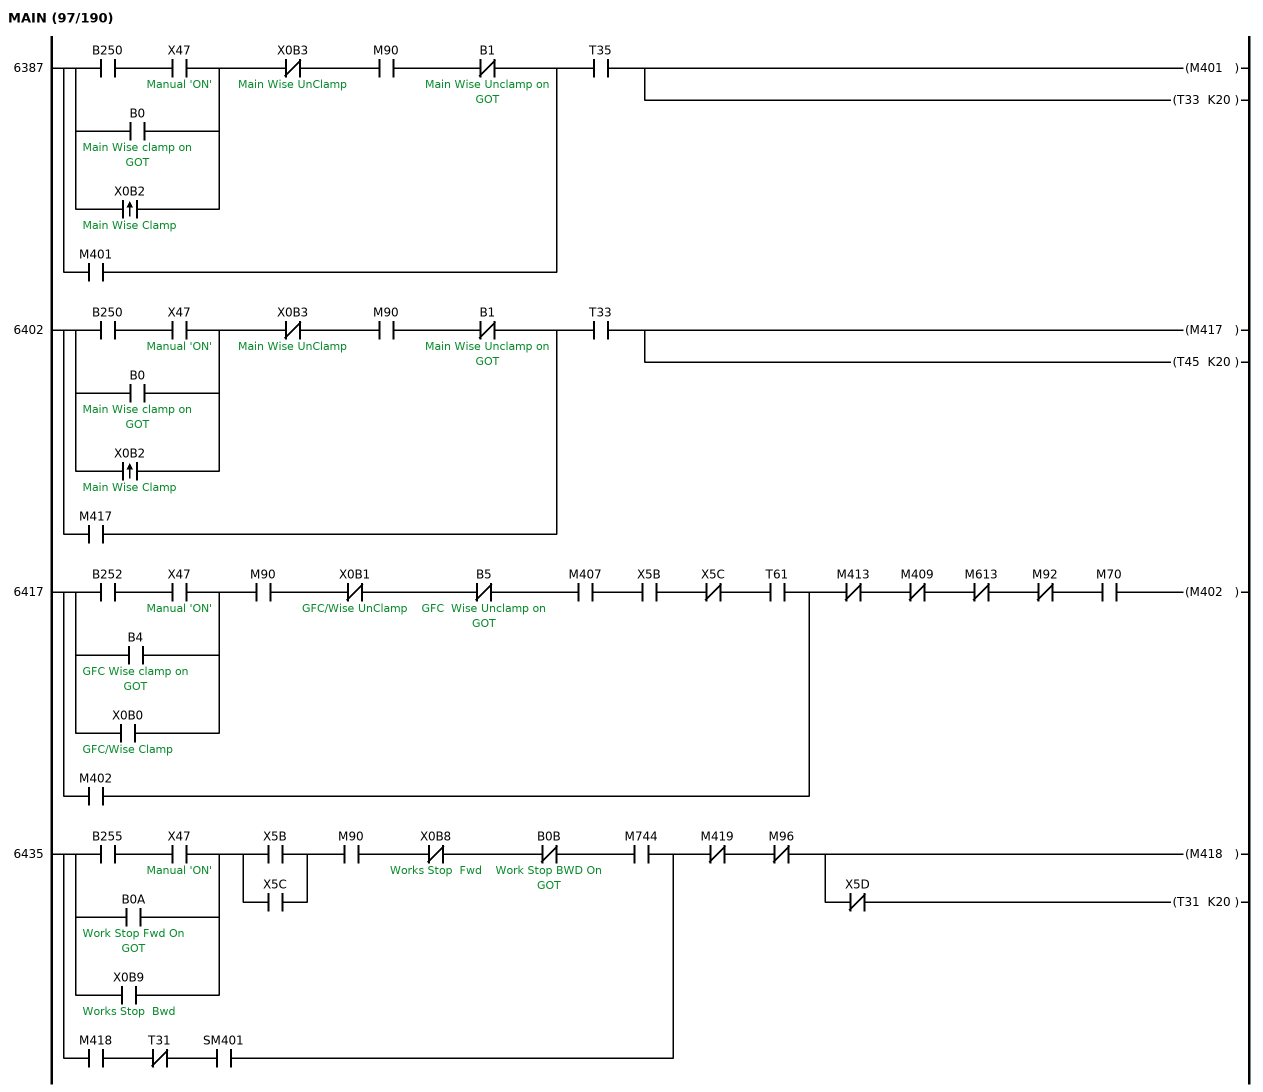
[picture p96: ladder of MAIN, rungs at steps 6387 to 6435]
6387  LD      B250
      AND     X47  ; Manual 'ON'
      OR      B0  ; Main Wise clamp on GOT
      ORP     X0B2  ; Main Wise Clamp
      ANI     X0B3  ; Main Wise UnClamp
      AND     M90
      ANI     B1  ; Main Wise Unclamp on GOT
      OR      M401
      AND     T35
      OUT     M401
      OUT     T33 K20
6402  LD      B250
      AND     X47  ; Manual 'ON'
      OR      B0  ; Main Wise clamp on GOT
      ORP     X0B2  ; Main Wise Clamp
      ANI     X0B3  ; Main Wise UnClamp
      AND     M90
      ANI     B1  ; Main Wise Unclamp on GOT
      OR      M417
      AND     T33
      OUT     M417
      OUT     T45 K20
6417  LD      B252
      AND     X47  ; Manual 'ON'
      OR      B4  ; GFC Wise clamp on GOT
      OR      X0B0  ; GFC/Wise Clamp
      AND     M90
      ANI     X0B1  ; GFC/Wise UnClamp
      ANI     B5  ; GFC  Wise Unclamp on GOT
      AND     M407
      AND     X5B
      ANI     X5C
      AND     T61
      OR      M402
      ANI     M413
      ANI     M409
      ANI     M613
      ANI     M92
      AND     M70
      OUT     M402
6435  LD      B255
      AND     X47  ; Manual 'ON'
      OR      B0A  ; Work Stop Fwd On GOT
      OR      X0B9  ; Works Stop  Bwd
      LD      X5B
      OR      X5C
      ANB
      AND     M90
      ANI     X0B8  ; Works Stop  Fwd
      ANI     B0B  ; Work Stop BWD On GOT
      AND     M744
      LD      M418
      ANI     T31
      AND     SM401
      ORB
      ANI     M419
      ANI     M96
      OUT     M418
      ANI     X5D
      OUT     T31 K20
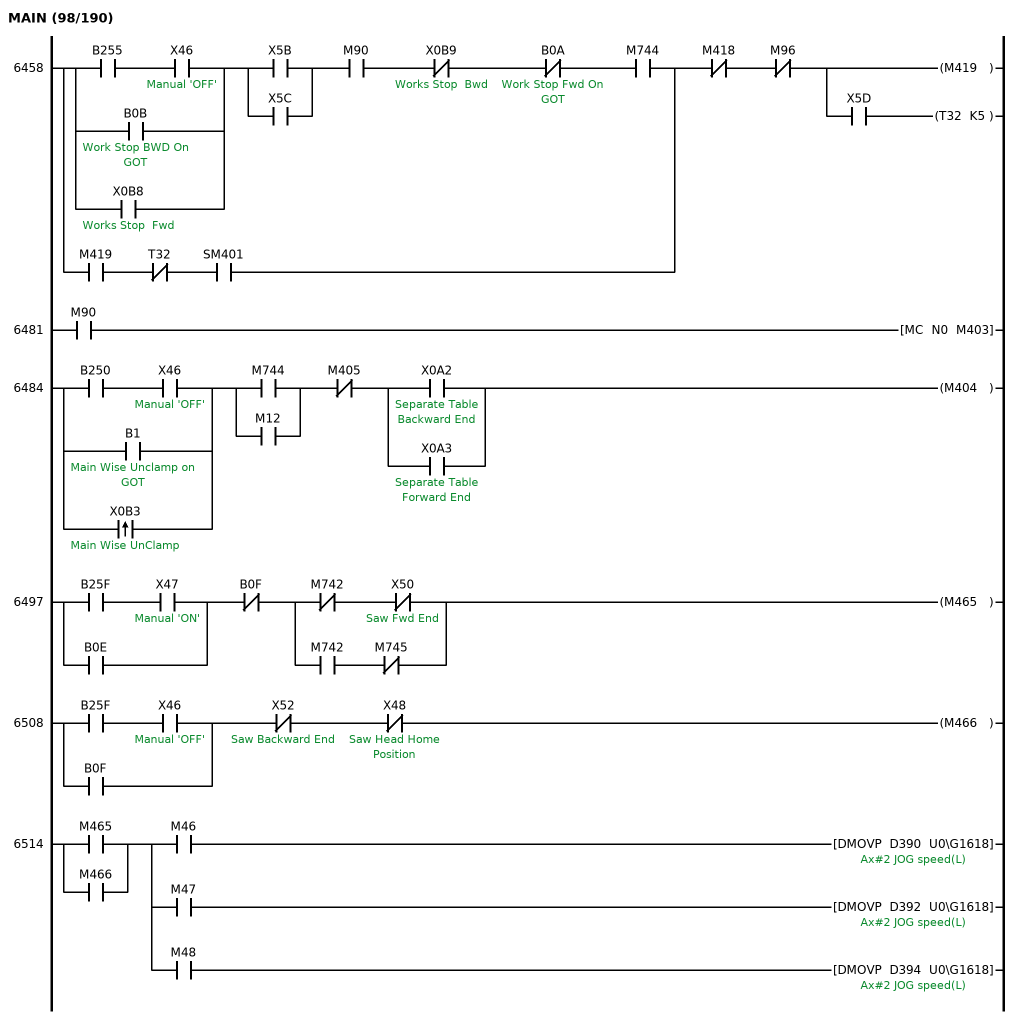
6458  LD      B255
      AND     X46  ; Manual 'OFF'
      OR      B0B  ; Work Stop BWD On GOT
      OR      X0B8  ; Works Stop  Fwd
      LD      X5B
      OR      X5C
      ANB
      AND     M90
      ANI     X0B9  ; Works Stop  Bwd
      ANI     B0A  ; Work Stop Fwd On GOT
      AND     M744
      LD      M419
      ANI     T32
      AND     SM401
      ORB
      ANI     M418
      ANI     M96
      OUT     M419
      AND     X5D
      OUT     T32 K5
6481  LD      M90
      MC      N0 M403
6484  LD      B250
      AND     X46  ; Manual 'OFF'
      OR      B1  ; Main Wise Unclamp on GOT
      ORP     X0B3  ; Main Wise UnClamp
      LD      M744
      OR      M12
      ANB
      ANI     M405
      LD      X0A2  ; Separate Table Backward End
      OR      X0A3  ; Separate Table Forward End
      ANB
      OUT     M404
6497  LD      B25F
      AND     X47  ; Manual 'ON'
      OR      B0E
      ANI     B0F
      LDI     M742
      ANI     X50  ; Saw Fwd End
      LD      M742
      ANI     M745
      ORB
      ANB
      OUT     M465
6508  LD      B25F
      AND     X46  ; Manual 'OFF'
      OR      B0F
      ANI     X52  ; Saw Backward End
      ANI     X48  ; Saw Head Home Position
      OUT     M466
6514  LD      M465
      OR      M466
      MPS
      AND     M46
      DMOVP   D390 U0\G1618
      MRD
      AND     M47
      DMOVP   D392 U0\G1618
      MPP
      AND     M48
      DMOVP   D394 U0\G1618
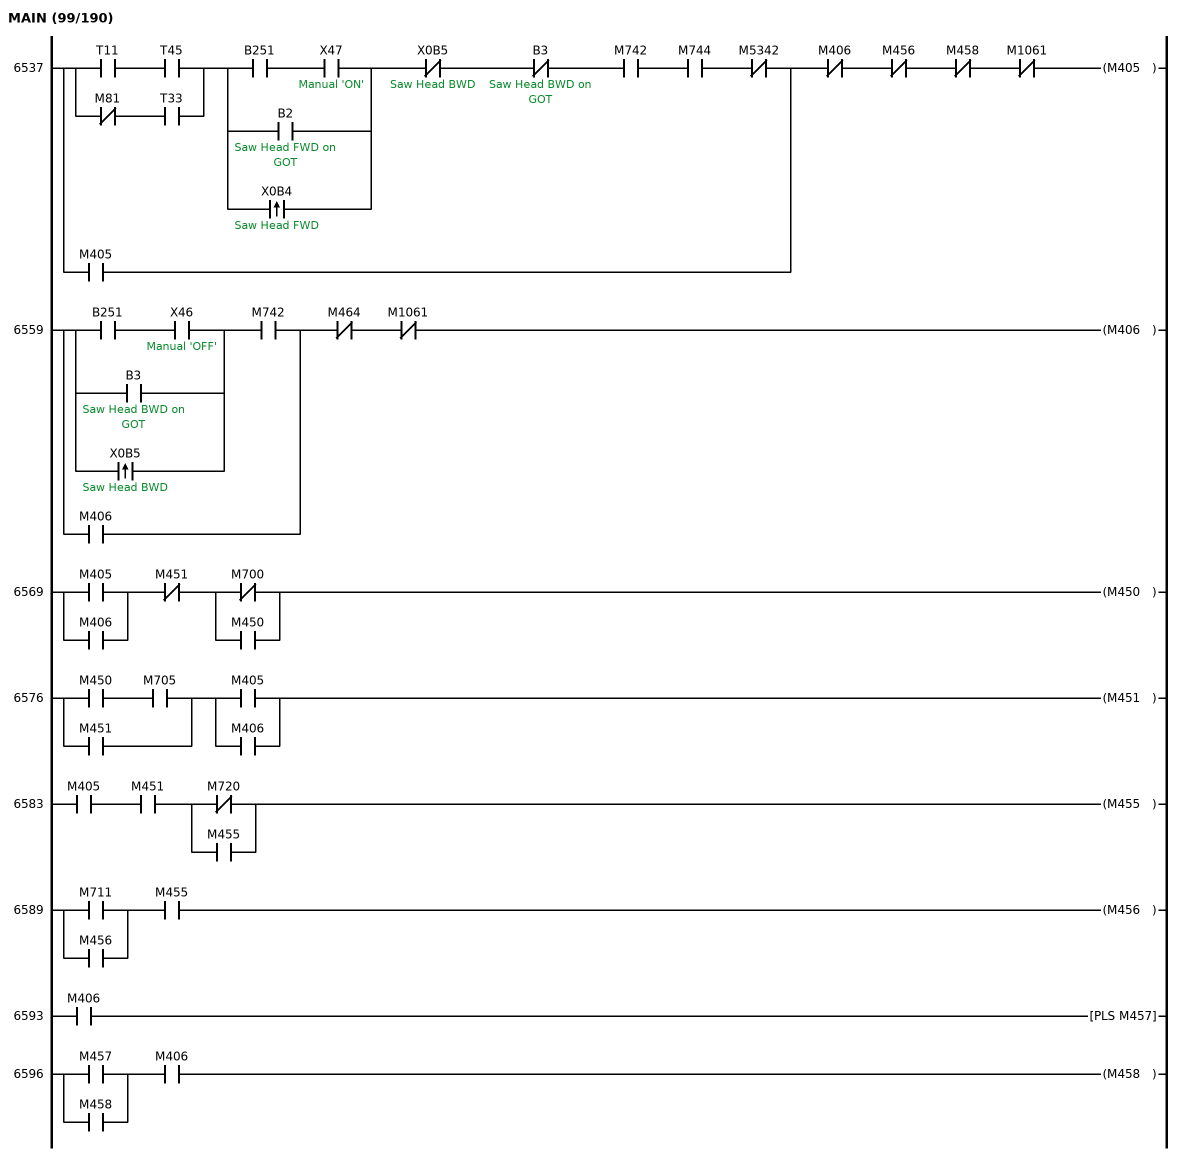
6537  LD      T11
      AND     T45
      LDI     M81
      AND     T33
      ORB
      LD      B251
      AND     X47  ; Manual 'ON'
      OR      B2  ; Saw Head FWD on GOT
      ORP     X0B4  ; Saw Head FWD
      ANB
      ANI     X0B5  ; Saw Head BWD
      ANI     B3  ; Saw Head BWD on GOT
      AND     M742
      AND     M744
      ANI     M5342
      OR      M405
      ANI     M406
      ANI     M456
      ANI     M458
      ANI     M1061
      OUT     M405
6559  LD      B251
      AND     X46  ; Manual 'OFF'
      OR      B3  ; Saw Head BWD on GOT
      ORP     X0B5  ; Saw Head BWD
      AND     M742
      OR      M406
      ANI     M464
      ANI     M1061
      OUT     M406
6569  LD      M405
      OR      M406
      ANI     M451
      LDI     M700
      OR      M450
      ANB
      OUT     M450
6576  LD      M450
      AND     M705
      OR      M451
      LD      M405
      OR      M406
      ANB
      OUT     M451
6583  LD      M405
      AND     M451
      LDI     M720
      OR      M455
      ANB
      OUT     M455
6589  LD      M711
      OR      M456
      AND     M455
      OUT     M456
6593  LD      M406
      PLS     M457
6596  LD      M457
      OR      M458
      AND     M406
      OUT     M458
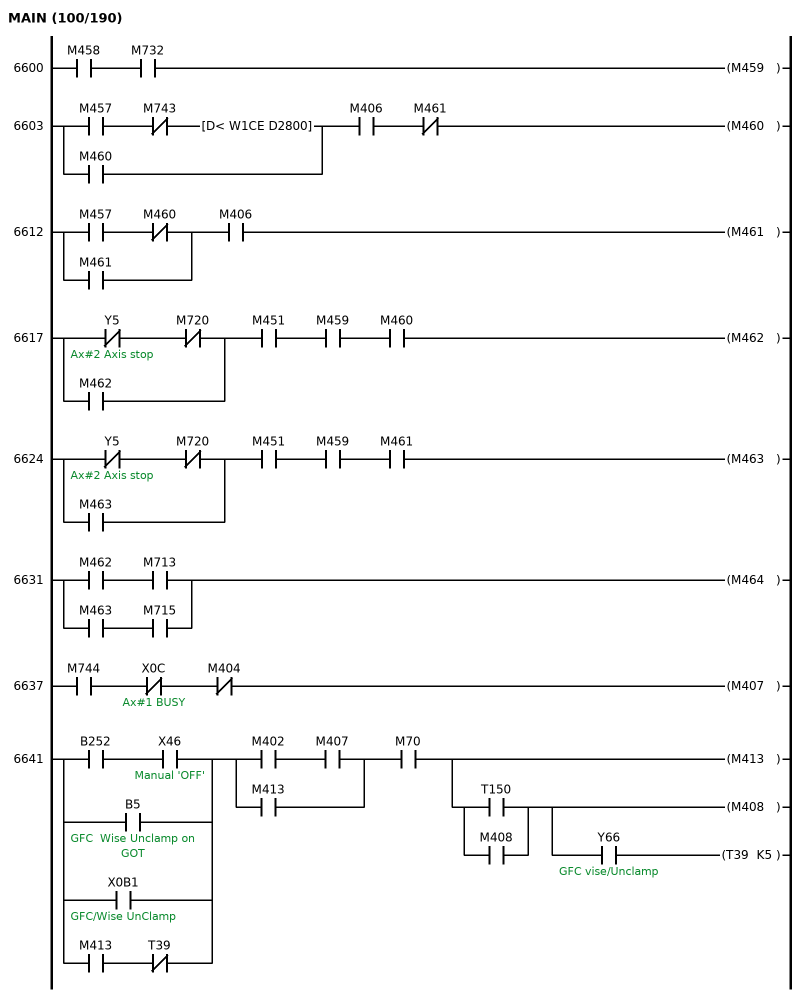
6600  LD      M458
      AND     M732
      OUT     M459
6603  LD      M457
      ANI     M743
      ANDD<   W1CE D2800
      OR      M460
      AND     M406
      ANI     M461
      OUT     M460
6612  LD      M457
      ANI     M460
      OR      M461
      AND     M406
      OUT     M461
6617  LDI     Y5  ; Ax#2 Axis stop
      ANI     M720
      OR      M462
      AND     M451
      AND     M459
      AND     M460
      OUT     M462
6624  LDI     Y5  ; Ax#2 Axis stop
      ANI     M720
      OR      M463
      AND     M451
      AND     M459
      AND     M461
      OUT     M463
6631  LD      M462
      AND     M713
      LD      M463
      AND     M715
      ORB
      OUT     M464
6637  LD      M744
      ANI     X0C  ; Ax#1 BUSY
      ANI     M404
      OUT     M407
6641  LD      B252
      AND     X46  ; Manual 'OFF'
      OR      B5  ; GFC  Wise Unclamp on GOT
      OR      X0B1  ; GFC/Wise UnClamp
      LD      M413
      ANI     T39
      ORB
      LD      M402
      AND     M407
      OR      M413
      ANB
      AND     M70
      OUT     M413
      LD      T150
      OR      M408
      ANB
      OUT     M408
      AND     Y66  ; GFC vise/Unclamp
      OUT     T39 K5
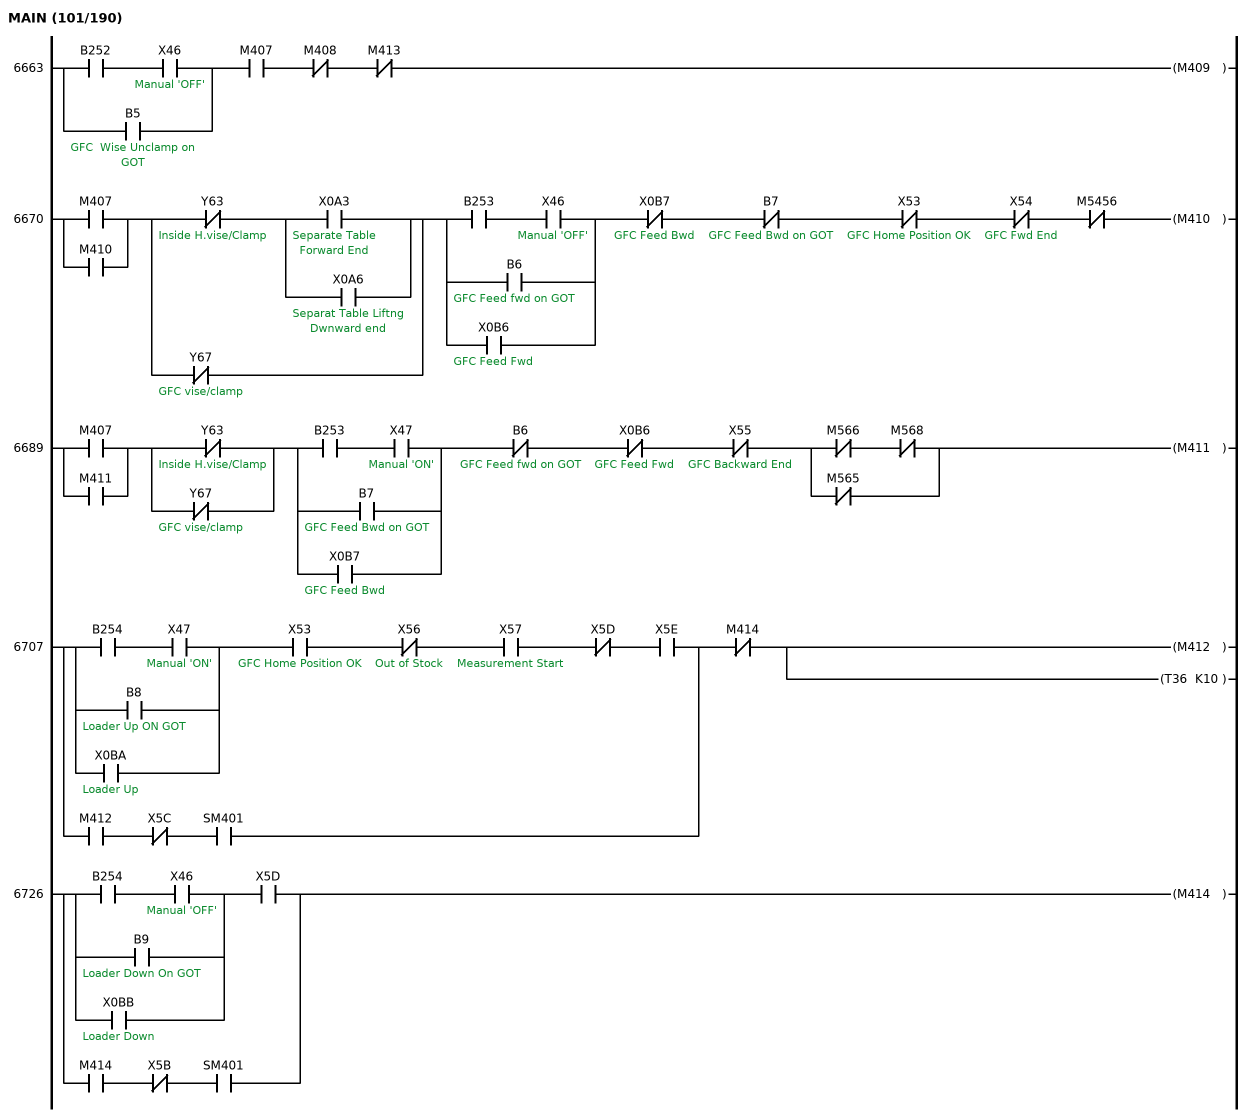
6663  LD      B252
      AND     X46  ; Manual 'OFF'
      OR      B5  ; GFC  Wise Unclamp on GOT
      AND     M407
      ANI     M408
      ANI     M413
      OUT     M409
6670  LD      M407
      OR      M410
      LDI     Y63  ; Inside H.vise/Clamp
      LD      X0A3  ; Separate Table Forward End
      OR      X0A6  ; Separat Table Liftng Dwnward end
      ANB
      ORI     Y67  ; GFC vise/clamp
      ANB
      LD      B253
      AND     X46  ; Manual 'OFF'
      OR      B6  ; GFC Feed fwd on GOT
      OR      X0B6  ; GFC Feed Fwd
      ANB
      ANI     X0B7  ; GFC Feed Bwd
      ANI     B7  ; GFC Feed Bwd on GOT
      ANI     X53  ; GFC Home Position OK
      ANI     X54  ; GFC Fwd End
      ANI     M5456
      OUT     M410
6689  LD      M407
      OR      M411
      LDI     Y63  ; Inside H.vise/Clamp
      ORI     Y67  ; GFC vise/clamp
      ANB
      LD      B253
      AND     X47  ; Manual 'ON'
      OR      B7  ; GFC Feed Bwd on GOT
      OR      X0B7  ; GFC Feed Bwd
      ANB
      ANI     B6  ; GFC Feed fwd on GOT
      ANI     X0B6  ; GFC Feed Fwd
      ANI     X55  ; GFC Backward End
      LDI     M566
      ANI     M568
      ORI     M565
      ANB
      OUT     M411
6707  LD      B254
      AND     X47  ; Manual 'ON'
      OR      B8  ; Loader Up ON GOT
      OR      X0BA  ; Loader Up
      AND     X53  ; GFC Home Position OK
      ANI     X56  ; Out of Stock
      AND     X57  ; Measurement Start
      ANI     X5D
      AND     X5E
      LD      M412
      ANI     X5C
      AND     SM401
      ORB
      ANI     M414
      OUT     M412
      OUT     T36 K10
6726  LD      B254
      AND     X46  ; Manual 'OFF'
      OR      B9  ; Loader Down On GOT
      OR      X0BB  ; Loader Down
      AND     X5D
      LD      M414
      ANI     X5B
      AND     SM401
      ORB
      OUT     M414
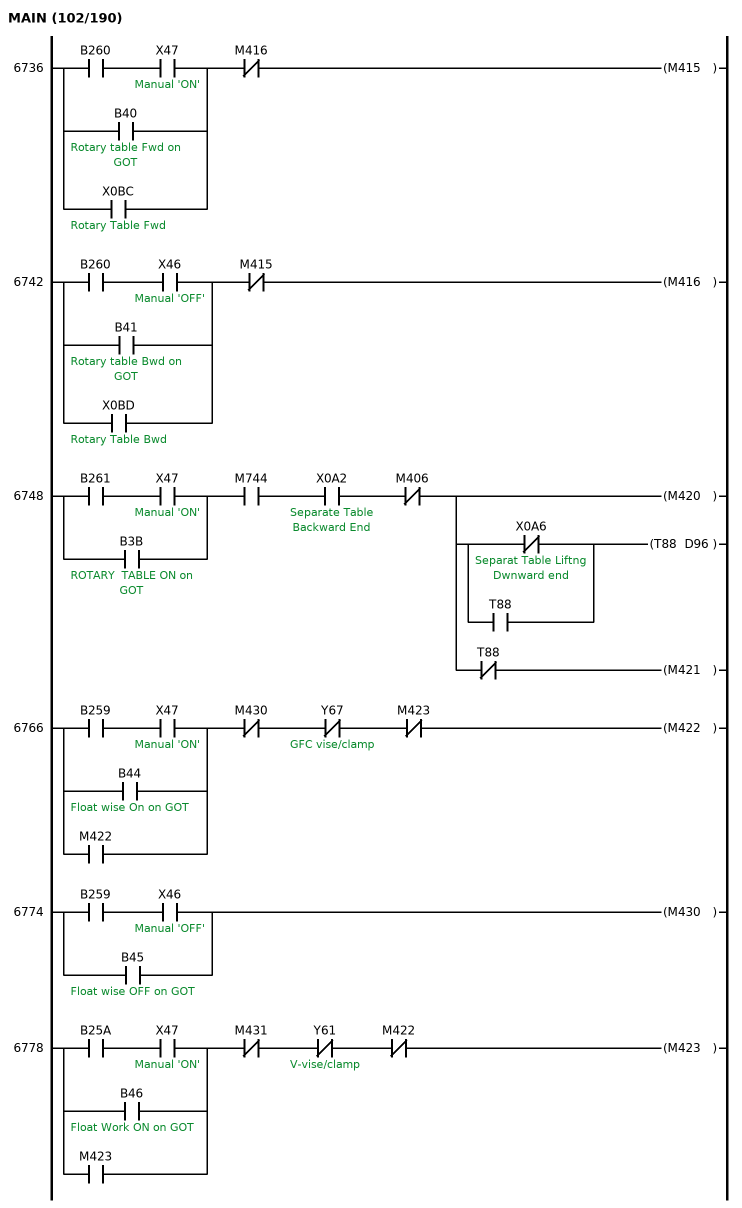
6736  LD      B260
      AND     X47  ; Manual 'ON'
      OR      B40  ; Rotary table Fwd on GOT
      OR      X0BC  ; Rotary Table Fwd
      ANI     M416
      OUT     M415
6742  LD      B260
      AND     X46  ; Manual 'OFF'
      OR      B41  ; Rotary table Bwd on GOT
      OR      X0BD  ; Rotary Table Bwd
      ANI     M415
      OUT     M416
6748  LD      B261
      AND     X47  ; Manual 'ON'
      OR      B3B  ; ROTARY  TABLE ON on GOT
      AND     M744
      AND     X0A2  ; Separate Table Backward End
      ANI     M406
      OUT     M420
      MPS
      LDI     X0A6  ; Separat Table Liftng Dwnward end
      OR      T88
      ANB
      OUT     T88 D96
      MPP
      ANI     T88
      OUT     M421
6766  LD      B259
      AND     X47  ; Manual 'ON'
      OR      B44  ; Float wise On on GOT
      OR      M422
      ANI     M430
      ANI     Y67  ; GFC vise/clamp
      ANI     M423
      OUT     M422
6774  LD      B259
      AND     X46  ; Manual 'OFF'
      OR      B45  ; Float wise OFF on GOT
      OUT     M430
6778  LD      B25A
      AND     X47  ; Manual 'ON'
      OR      B46  ; Float Work ON on GOT
      OR      M423
      ANI     M431
      ANI     Y61  ; V-vise/clamp
      ANI     M422
      OUT     M423
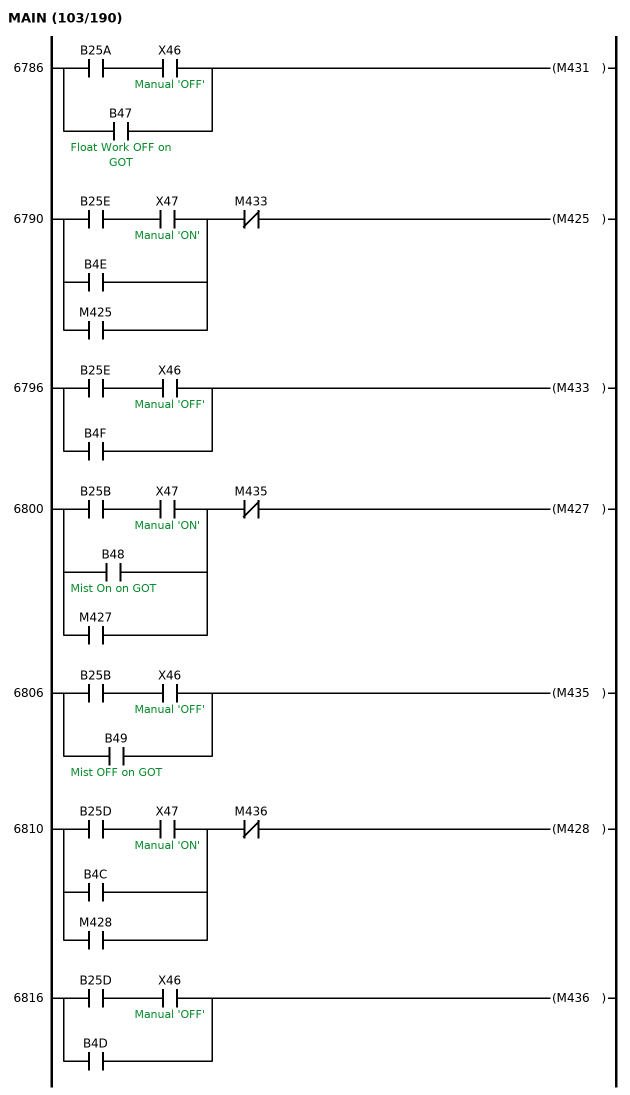
6786  LD      B25A
      AND     X46  ; Manual 'OFF'
      OR      B47  ; Float Work OFF on GOT
      OUT     M431
6790  LD      B25E
      AND     X47  ; Manual 'ON'
      OR      B4E
      OR      M425
      ANI     M433
      OUT     M425
6796  LD      B25E
      AND     X46  ; Manual 'OFF'
      OR      B4F
      OUT     M433
6800  LD      B25B
      AND     X47  ; Manual 'ON'
      OR      B48  ; Mist On on GOT
      OR      M427
      ANI     M435
      OUT     M427
6806  LD      B25B
      AND     X46  ; Manual 'OFF'
      OR      B49  ; Mist OFF on GOT
      OUT     M435
6810  LD      B25D
      AND     X47  ; Manual 'ON'
      OR      B4C
      OR      M428
      ANI     M436
      OUT     M428
6816  LD      B25D
      AND     X46  ; Manual 'OFF'
      OR      B4D
      OUT     M436
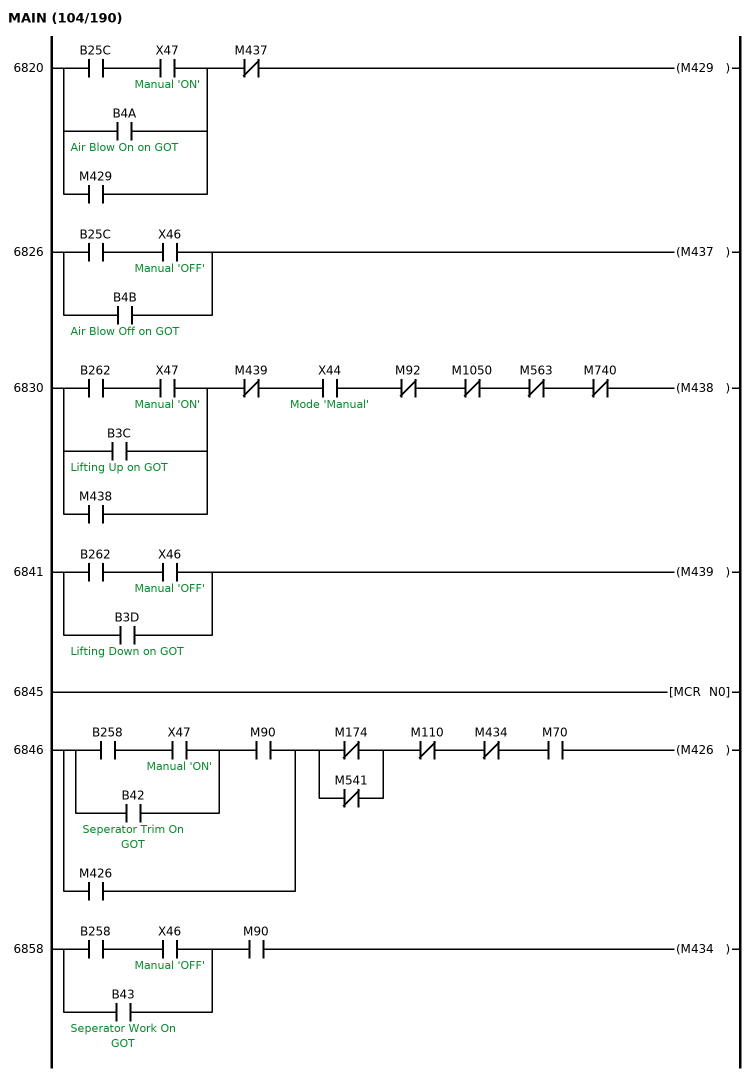
6820  LD      B25C
      AND     X47  ; Manual 'ON'
      OR      B4A  ; Air Blow On on GOT
      OR      M429
      ANI     M437
      OUT     M429
6826  LD      B25C
      AND     X46  ; Manual 'OFF'
      OR      B4B  ; Air Blow Off on GOT
      OUT     M437
6830  LD      B262
      AND     X47  ; Manual 'ON'
      OR      B3C  ; Lifting Up on GOT
      OR      M438
      ANI     M439
      AND     X44  ; Mode 'Manual'
      ANI     M92
      ANI     M1050
      ANI     M563
      ANI     M740
      OUT     M438
6841  LD      B262
      AND     X46  ; Manual 'OFF'
      OR      B3D  ; Lifting Down on GOT
      OUT     M439
6845  MCR     N0
6846  LD      B258
      AND     X47  ; Manual 'ON'
      OR      B42  ; Seperator Trim On GOT
      AND     M90
      OR      M426
      LDI     M174
      ORI     M541
      ANB
      ANI     M110
      ANI     M434
      AND     M70
      OUT     M426
6858  LD      B258
      AND     X46  ; Manual 'OFF'
      OR      B43  ; Seperator Work On GOT
      AND     M90
      OUT     M434
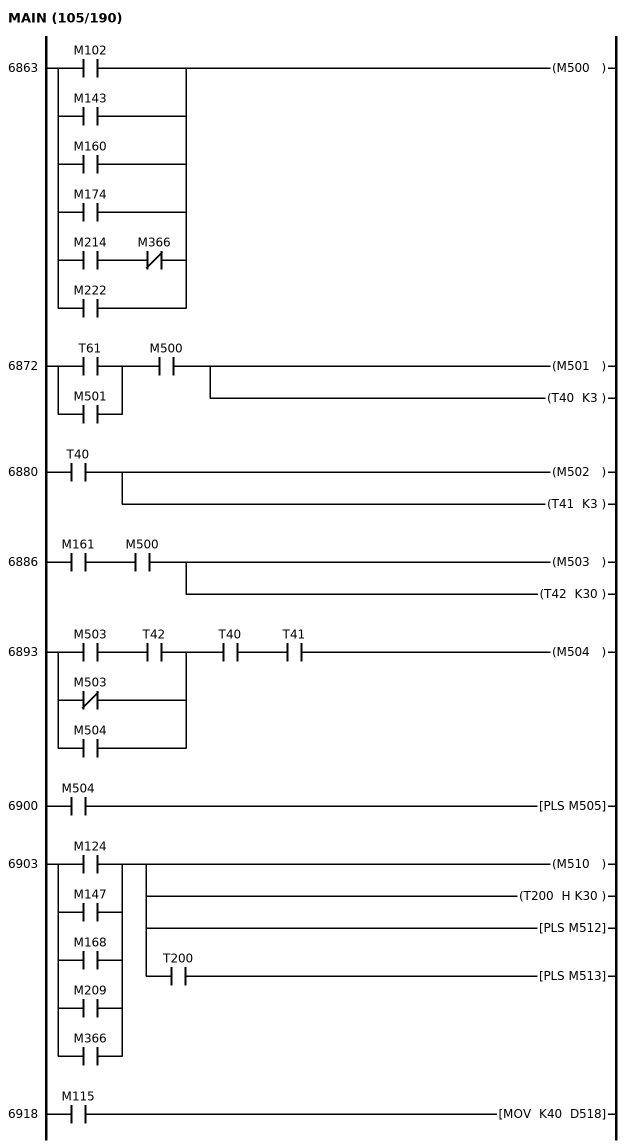
6863  LD      M102
      OR      M143
      OR      M160
      OR      M174
      LD      M214
      ANI     M366
      ORB
      OR      M222
      OUT     M500
6872  LD      T61
      OR      M501
      AND     M500
      OUT     M501
      OUT     T40 K3
6880  LD      T40
      OUT     M502
      OUT     T41 K3
6886  LD      M161
      AND     M500
      OUT     M503
      OUT     T42 K30
6893  LD      M503
      AND     T42
      ORI     M503
      OR      M504
      AND     T40
      AND     T41
      OUT     M504
6900  LD      M504
      PLS     M505
6903  LD      M124
      OR      M147
      OR      M168
      OR      M209
      OR      M366
      OUT     M510
      OUTH    T200 K30
      PLS     M512
      AND     T200
      PLS     M513
6918  LD      M115
      MOV     K40 D518
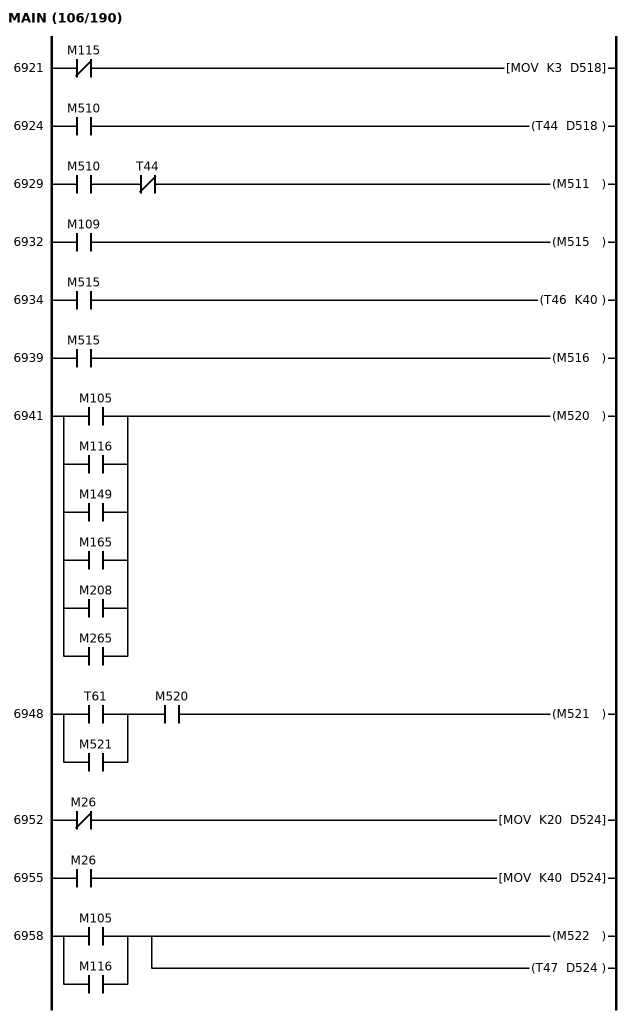
6921  LDI     M115
      MOV     K3 D518
6924  LD      M510
      OUT     T44 D518
6929  LD      M510
      ANI     T44
      OUT     M511
6932  LD      M109
      OUT     M515
6934  LD      M515
      OUT     T46 K40
6939  LD      M515
      OUT     M516
6941  LD      M105
      OR      M116
      OR      M149
      OR      M165
      OR      M208
      OR      M265
      OUT     M520
6948  LD      T61
      OR      M521
      AND     M520
      OUT     M521
6952  LDI     M26
      MOV     K20 D524
6955  LD      M26
      MOV     K40 D524
6958  LD      M105
      OR      M116
      OUT     M522
      OUT     T47 D524
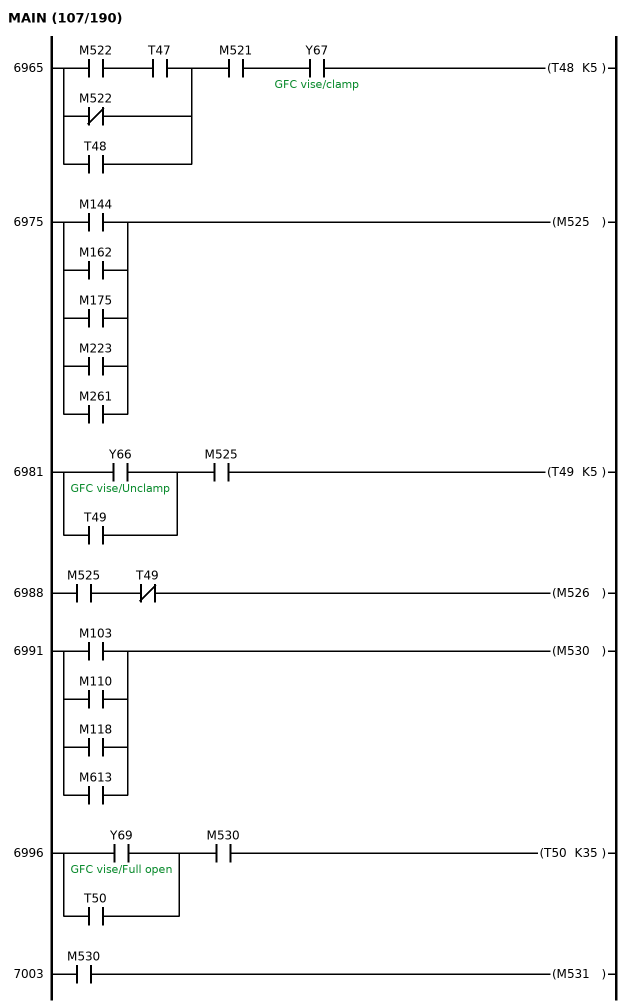
6965  LD      M522
      AND     T47
      ORI     M522
      OR      T48
      AND     M521
      AND     Y67  ; GFC vise/clamp
      OUT     T48 K5
6975  LD      M144
      OR      M162
      OR      M175
      OR      M223
      OR      M261
      OUT     M525
6981  LD      Y66  ; GFC vise/Unclamp
      OR      T49
      AND     M525
      OUT     T49 K5
6988  LD      M525
      ANI     T49
      OUT     M526
6991  LD      M103
      OR      M110
      OR      M118
      OR      M613
      OUT     M530
6996  LD      Y69  ; GFC vise/Full open
      OR      T50
      AND     M530
      OUT     T50 K35
7003  LD      M530
      OUT     M531
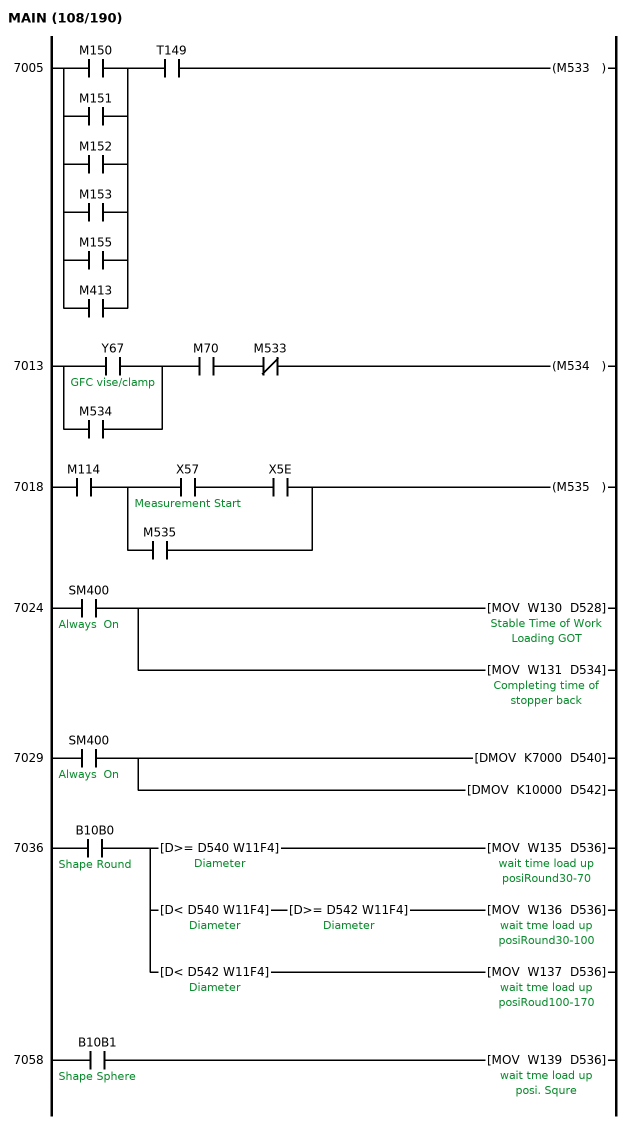
7005  LD      M150
      OR      M151
      OR      M152
      OR      M153
      OR      M155
      OR      M413
      AND     T149
      OUT     M533
7013  LD      Y67  ; GFC vise/clamp
      OR      M534
      AND     M70
      ANI     M533
      OUT     M534
7018  LD      M114
      LD      X57  ; Measurement Start
      AND     X5E
      OR      M535
      ANB
      OUT     M535
7024  LD      SM400  ; Always  On
      MOV     W130 D528
      MOV     W131 D534  ; Completing time of stopper back
7029  LD      SM400  ; Always  On
      DMOV    K7000 D540
      DMOV    K10000 D542
7036  LD      B10B0  ; Shape Round
      MPS
      ANDD>=  D540 W11F4  ; Diameter
      MOV     W135 D536  ; wait time load up posiRound30-70
      MRD
      ANDD<   D540 W11F4  ; Diameter
      ANDD>=  D542 W11F4  ; Diameter
      MOV     W136 D536  ; wait tme load up posiRound30-100
      MPP
      ANDD<   D542 W11F4  ; Diameter
      MOV     W137 D536  ; wait tme load up posiRoud100-170
7058  LD      B10B1  ; Shape Sphere
      MOV     W139 D536  ; wait tme load up posi. Squre
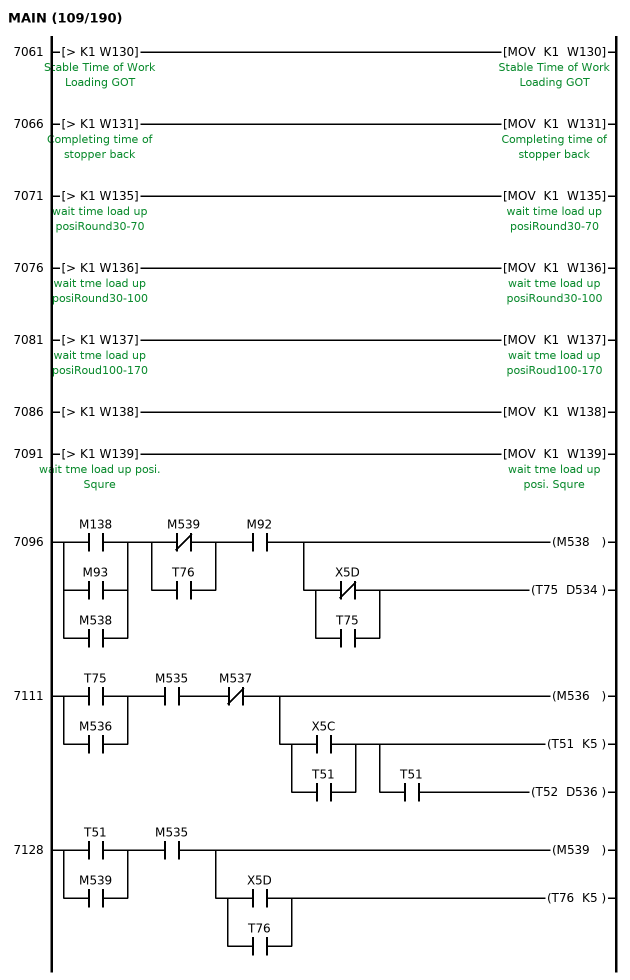
7061  LD>     K1 W130  ; Stable Time of Work Loading GOT
      MOV     K1 W130
7066  LD>     K1 W131  ; Completing time of stopper back
      MOV     K1 W131
7071  LD>     K1 W135  ; wait time load up posiRound30-70
      MOV     K1 W135
7076  LD>     K1 W136  ; wait tme load up posiRound30-100
      MOV     K1 W136
7081  LD>     K1 W137  ; wait tme load up posiRoud100-170
      MOV     K1 W137
7086  LD>     K1 W138
      MOV     K1 W138
7091  LD>     K1 W139  ; wait tme load up posi. Squre
      MOV     K1 W139
7096  LD      M138
      OR      M93
      OR      M538
      LDI     M539
      OR      T76
      ANB
      AND     M92
      OUT     M538
      LDI     X5D
      OR      T75
      ANB
      OUT     T75 D534
7111  LD      T75
      OR      M536
      AND     M535
      ANI     M537
      OUT     M536
      LD      X5C
      OR      T51
      ANB
      OUT     T51 K5
      AND     T51
      OUT     T52 D536
7128  LD      T51
      OR      M539
      AND     M535
      OUT     M539
      LD      X5D
      OR      T76
      ANB
      OUT     T76 K5
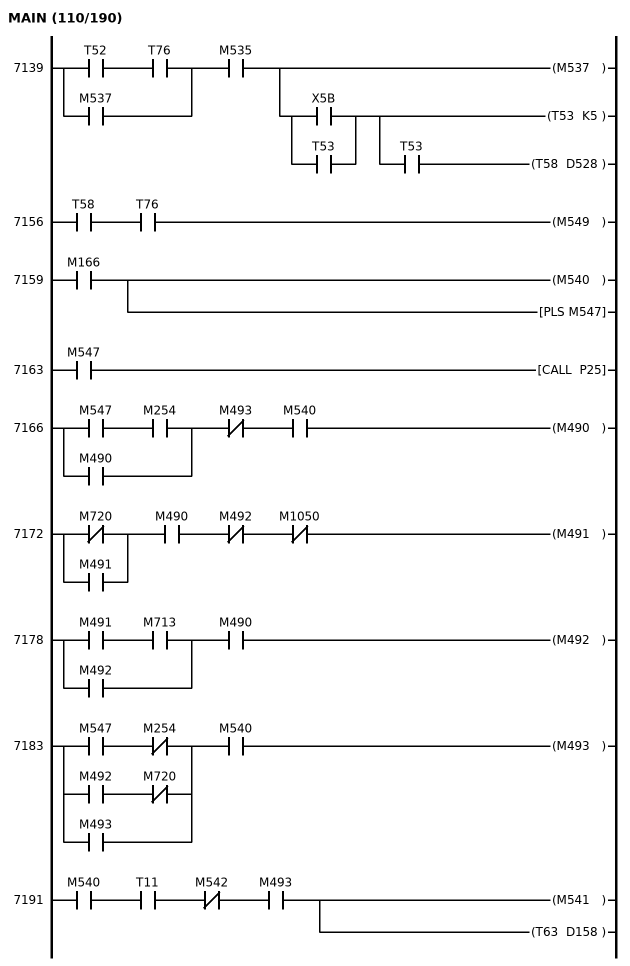
7139  LD      T52
      AND     T76
      OR      M537
      AND     M535
      OUT     M537
      LD      X5B
      OR      T53
      ANB
      OUT     T53 K5
      AND     T53
      OUT     T58 D528
7156  LD      T58
      AND     T76
      OUT     M549
7159  LD      M166
      OUT     M540
      PLS     M547
7163  LD      M547
      CALL    P25
7166  LD      M547
      AND     M254
      OR      M490
      ANI     M493
      AND     M540
      OUT     M490
7172  LDI     M720
      OR      M491
      AND     M490
      ANI     M492
      ANI     M1050
      OUT     M491
7178  LD      M491
      AND     M713
      OR      M492
      AND     M490
      OUT     M492
7183  LD      M547
      ANI     M254
      LD      M492
      ANI     M720
      ORB
      OR      M493
      AND     M540
      OUT     M493
7191  LD      M540
      AND     T11
      ANI     M542
      AND     M493
      OUT     M541
      OUT     T63 D158
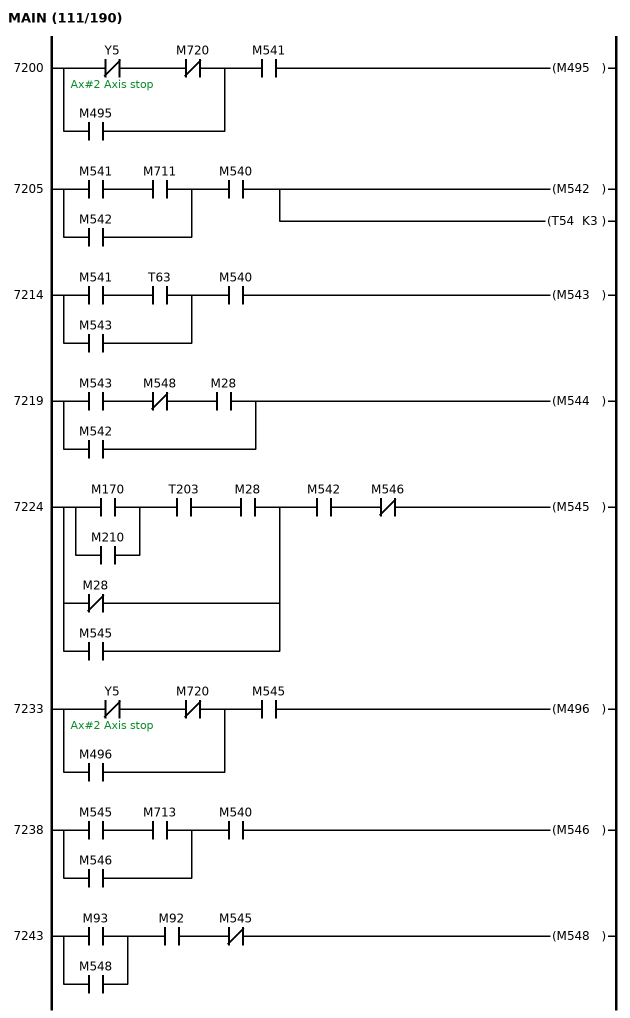
7200  LDI     Y5  ; Ax#2 Axis stop
      ANI     M720
      OR      M495
      AND     M541
      OUT     M495
7205  LD      M541
      AND     M711
      OR      M542
      AND     M540
      OUT     M542
      OUT     T54 K3
7214  LD      M541
      AND     T63
      OR      M543
      AND     M540
      OUT     M543
7219  LD      M543
      ANI     M548
      AND     M28
      OR      M542
      OUT     M544
7224  LD      M170
      OR      M210
      AND     T203
      AND     M28
      ORI     M28
      OR      M545
      AND     M542
      ANI     M546
      OUT     M545
7233  LDI     Y5  ; Ax#2 Axis stop
      ANI     M720
      OR      M496
      AND     M545
      OUT     M496
7238  LD      M545
      AND     M713
      OR      M546
      AND     M540
      OUT     M546
7243  LD      M93
      OR      M548
      AND     M92
      ANI     M545
      OUT     M548
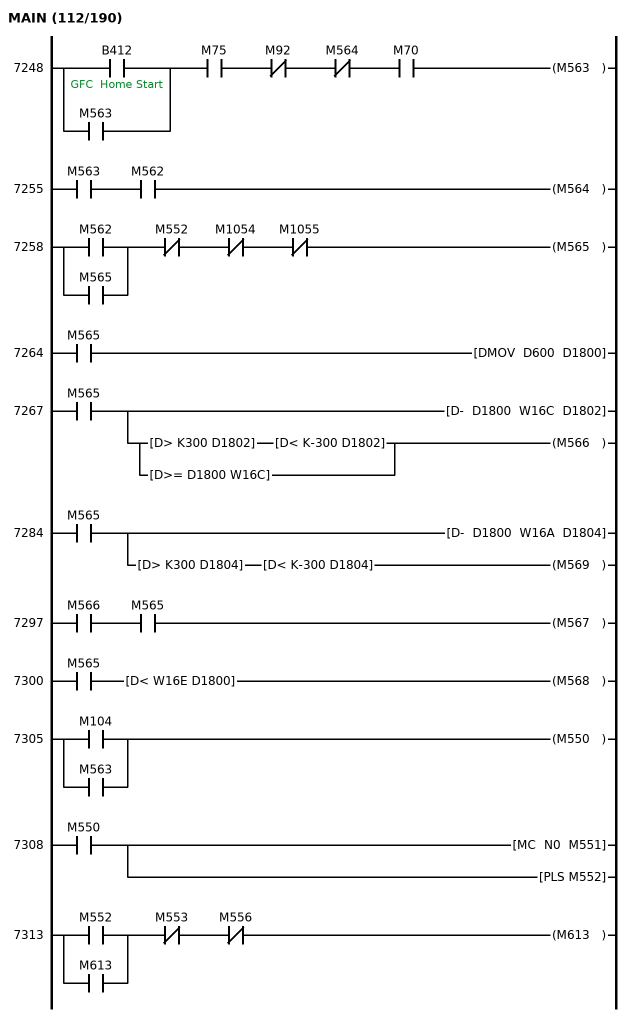
7248  LD      B412  ; GFC  Home Start
      OR      M563
      AND     M75
      ANI     M92
      ANI     M564
      AND     M70
      OUT     M563
7255  LD      M563
      AND     M562
      OUT     M564
7258  LD      M562
      OR      M565
      ANI     M552
      ANI     M1054
      ANI     M1055
      OUT     M565
7264  LD      M565
      DMOV    D600 D1800
7267  LD      M565
      D-      D1800 W16C D1802
      LDD>    K300 D1802
      ANDD<   K-300 D1802
      ORD>=   D1800 W16C
      ANB
      OUT     M566
7284  LD      M565
      D-      D1800 W16A D1804
      ANDD>   K300 D1804
      ANDD<   K-300 D1804
      OUT     M569
7297  LD      M566
      AND     M565
      OUT     M567
7300  LD      M565
      ANDD<   W16E D1800
      OUT     M568
7305  LD      M104
      OR      M563
      OUT     M550
7308  LD      M550
      MC      N0 M551
      PLS     M552
7313  LD      M552
      OR      M613
      ANI     M553
      ANI     M556
      OUT     M613
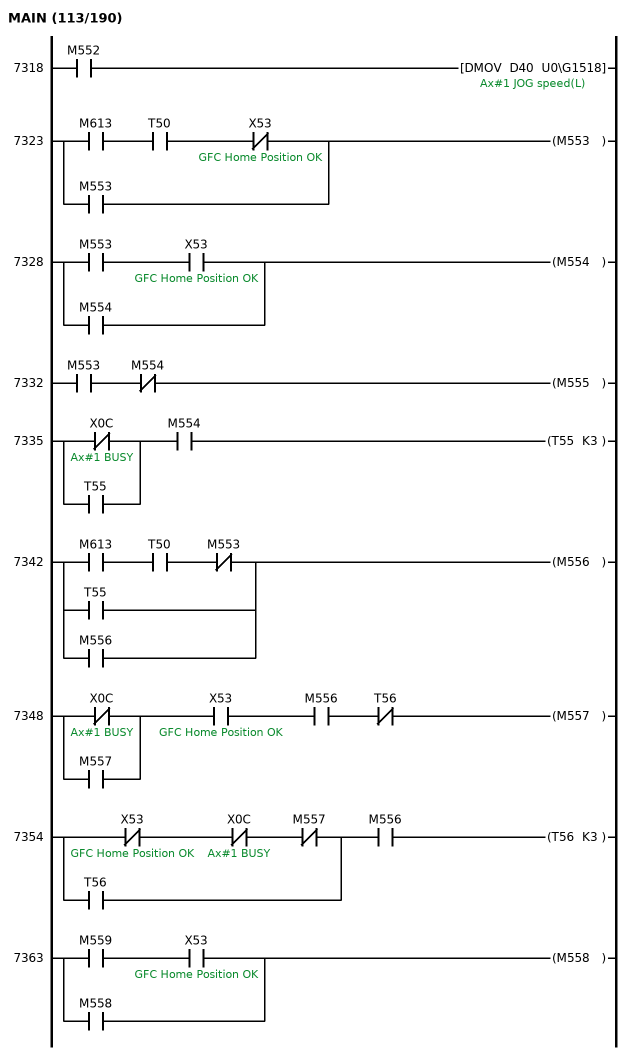
7318  LD      M552
      DMOV    D40 U0\G1518
7323  LD      M613
      AND     T50
      ANI     X53  ; GFC Home Position OK
      OR      M553
      OUT     M553
7328  LD      M553
      AND     X53  ; GFC Home Position OK
      OR      M554
      OUT     M554
7332  LD      M553
      ANI     M554
      OUT     M555
7335  LDI     X0C  ; Ax#1 BUSY
      OR      T55
      AND     M554
      OUT     T55 K3
7342  LD      M613
      AND     T50
      ANI     M553
      OR      T55
      OR      M556
      OUT     M556
7348  LDI     X0C  ; Ax#1 BUSY
      OR      M557
      AND     X53  ; GFC Home Position OK
      AND     M556
      ANI     T56
      OUT     M557
7354  LDI     X53  ; GFC Home Position OK
      ANI     X0C  ; Ax#1 BUSY
      ANI     M557
      OR      T56
      AND     M556
      OUT     T56 K3
7363  LD      M559
      AND     X53  ; GFC Home Position OK
      OR      M558
      OUT     M558
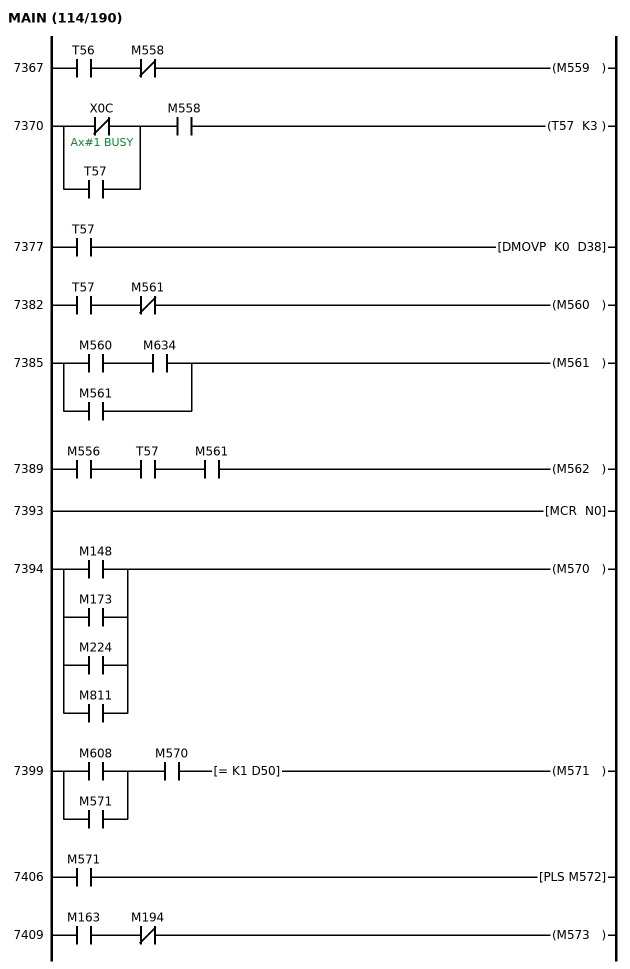
7367  LD      T56
      ANI     M558
      OUT     M559
7370  LDI     X0C  ; Ax#1 BUSY
      OR      T57
      AND     M558
      OUT     T57 K3
7377  LD      T57
      DMOVP   K0 D38
7382  LD      T57
      ANI     M561
      OUT     M560
7385  LD      M560
      AND     M634
      OR      M561
      OUT     M561
7389  LD      M556
      AND     T57
      AND     M561
      OUT     M562
7393  MCR     N0
7394  LD      M148
      OR      M173
      OR      M224
      OR      M811
      OUT     M570
7399  LD      M608
      OR      M571
      AND     M570
      AND=    K1 D50
      OUT     M571
7406  LD      M571
      PLS     M572
7409  LD      M163
      ANI     M194
      OUT     M573
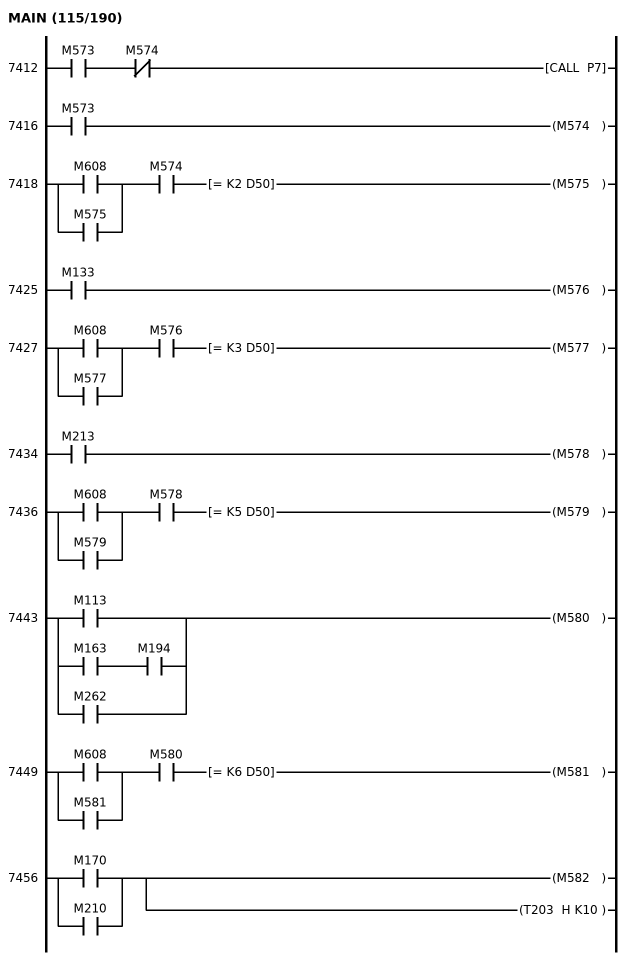
7412  LD      M573
      ANI     M574
      CALL    P7
7416  LD      M573
      OUT     M574
7418  LD      M608
      OR      M575
      AND     M574
      AND=    K2 D50
      OUT     M575
7425  LD      M133
      OUT     M576
7427  LD      M608
      OR      M577
      AND     M576
      AND=    K3 D50
      OUT     M577
7434  LD      M213
      OUT     M578
7436  LD      M608
      OR      M579
      AND     M578
      AND=    K5 D50
      OUT     M579
7443  LD      M113
      LD      M163
      AND     M194
      ORB
      OR      M262
      OUT     M580
7449  LD      M608
      OR      M581
      AND     M580
      AND=    K6 D50
      OUT     M581
7456  LD      M170
      OR      M210
      OUT     M582
      OUTH    T203 K10
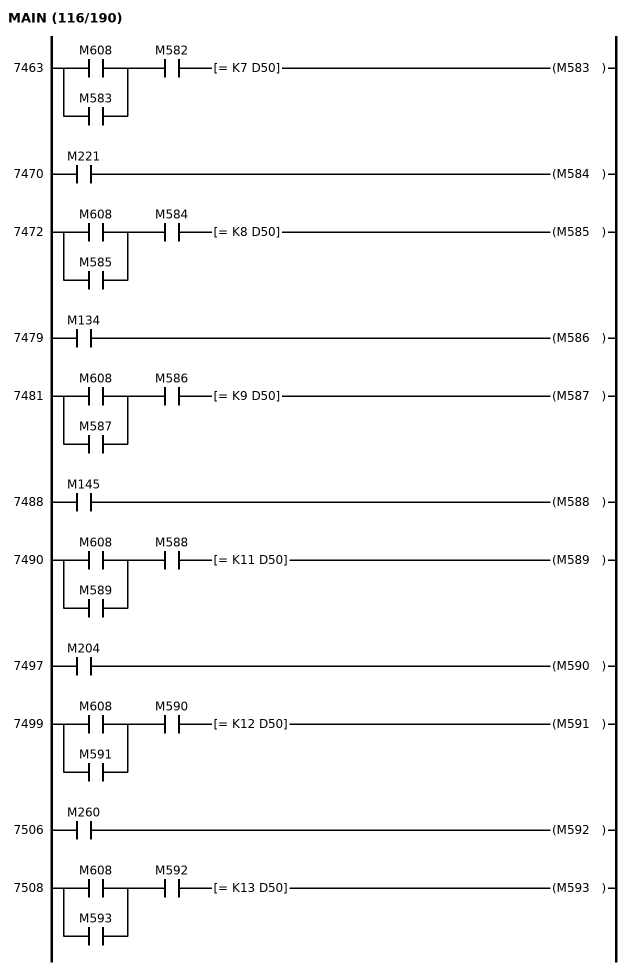
7463  LD      M608
      OR      M583
      AND     M582
      AND=    K7 D50
      OUT     M583
7470  LD      M221
      OUT     M584
7472  LD      M608
      OR      M585
      AND     M584
      AND=    K8 D50
      OUT     M585
7479  LD      M134
      OUT     M586
7481  LD      M608
      OR      M587
      AND     M586
      AND=    K9 D50
      OUT     M587
7488  LD      M145
      OUT     M588
7490  LD      M608
      OR      M589
      AND     M588
      AND=    K11 D50
      OUT     M589
7497  LD      M204
      OUT     M590
7499  LD      M608
      OR      M591
      AND     M590
      AND=    K12 D50
      OUT     M591
7506  LD      M260
      OUT     M592
7508  LD      M608
      OR      M593
      AND     M592
      AND=    K13 D50
      OUT     M593
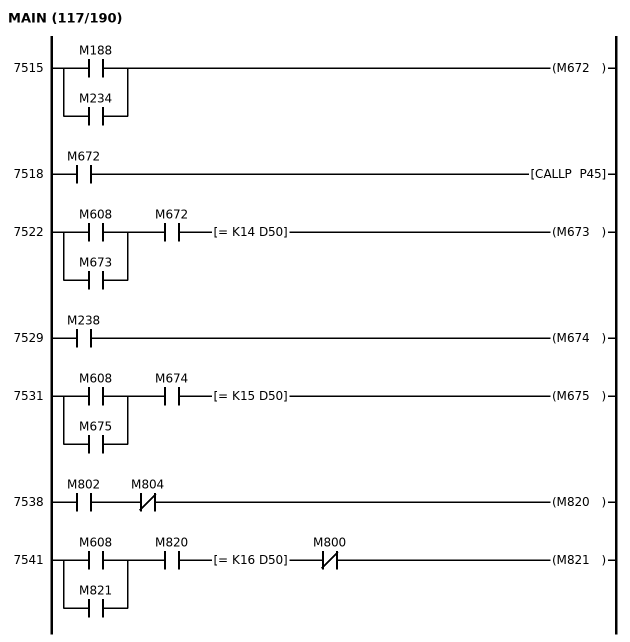
7515  LD      M188
      OR      M234
      OUT     M672
7518  LD      M672
      CALLP   P45
7522  LD      M608
      OR      M673
      AND     M672
      AND=    K14 D50
      OUT     M673
7529  LD      M238
      OUT     M674
7531  LD      M608
      OR      M675
      AND     M674
      AND=    K15 D50
      OUT     M675
7538  LD      M802
      ANI     M804
      OUT     M820
7541  LD      M608
      OR      M821
      AND     M820
      AND=    K16 D50
      ANI     M800
      OUT     M821
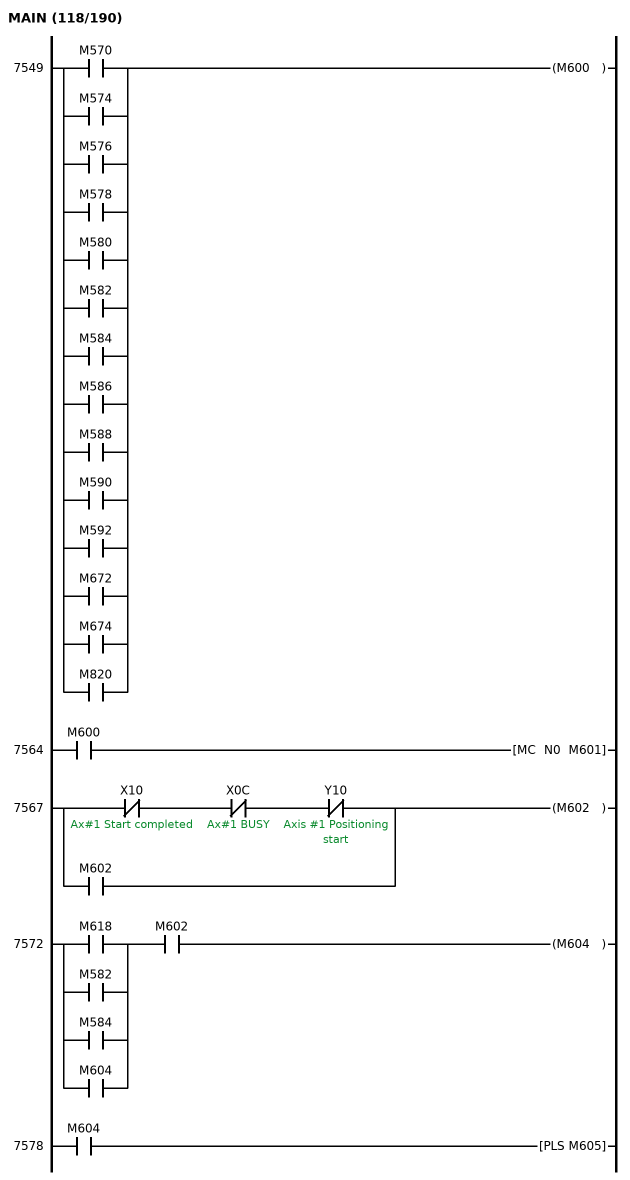
7549  LD      M570
      OR      M574
      OR      M576
      OR      M578
      OR      M580
      OR      M582
      OR      M584
      OR      M586
      OR      M588
      OR      M590
      OR      M592
      OR      M672
      OR      M674
      OR      M820
      OUT     M600
7564  LD      M600
      MC      N0 M601
7567  LDI     X10  ; Ax#1 Start completed
      ANI     X0C  ; Ax#1 BUSY
      ANI     Y10  ; Axis #1 Positioning start
      OR      M602
      OUT     M602
7572  LD      M618
      OR      M582
      OR      M584
      OR      M604
      AND     M602
      OUT     M604
7578  LD      M604
      PLS     M605
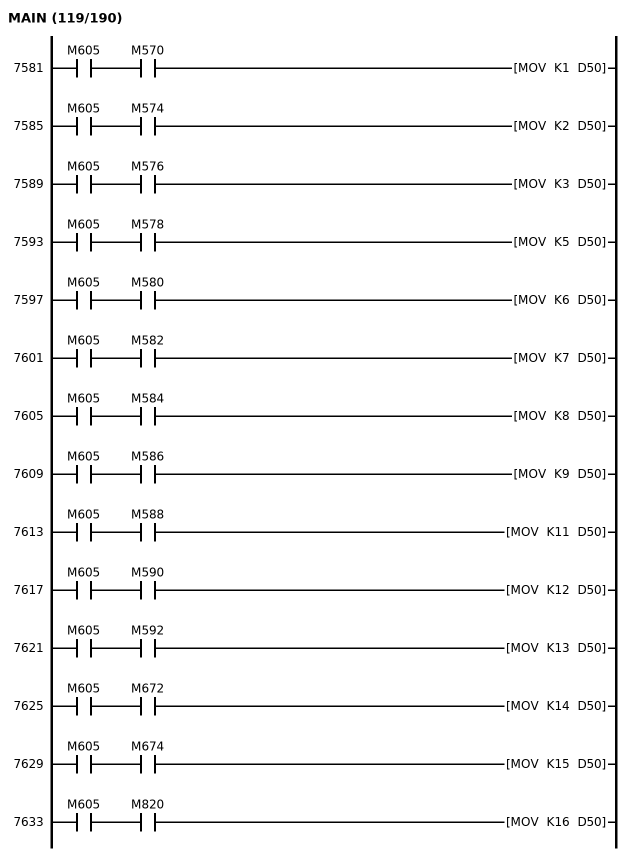
7581  LD      M605
      AND     M570
      MOV     K1 D50
7585  LD      M605
      AND     M574
      MOV     K2 D50
7589  LD      M605
      AND     M576
      MOV     K3 D50
7593  LD      M605
      AND     M578
      MOV     K5 D50
7597  LD      M605
      AND     M580
      MOV     K6 D50
7601  LD      M605
      AND     M582
      MOV     K7 D50
7605  LD      M605
      AND     M584
      MOV     K8 D50
7609  LD      M605
      AND     M586
      MOV     K9 D50
7613  LD      M605
      AND     M588
      MOV     K11 D50
7617  LD      M605
      AND     M590
      MOV     K12 D50
7621  LD      M605
      AND     M592
      MOV     K13 D50
7625  LD      M605
      AND     M672
      MOV     K14 D50
7629  LD      M605
      AND     M674
      MOV     K15 D50
7633  LD      M605
      AND     M820
      MOV     K16 D50
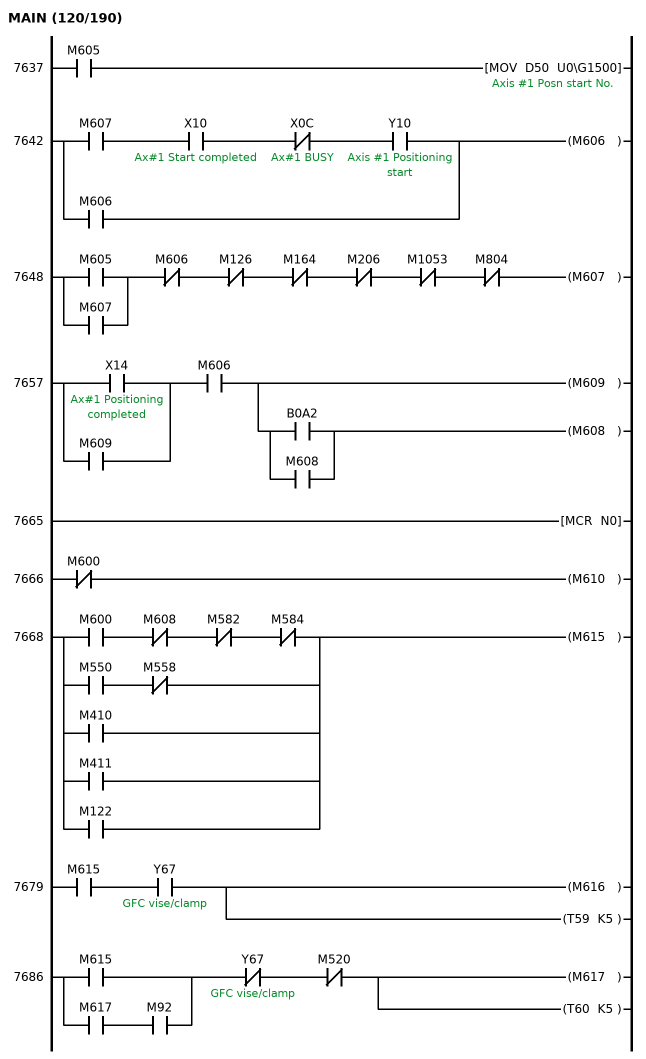
7637  LD      M605
      MOV     D50 U0\G1500  ; Axis #1 Posn start No.
7642  LD      M607
      AND     X10  ; Ax#1 Start completed
      ANI     X0C  ; Ax#1 BUSY
      AND     Y10  ; Axis #1 Positioning start
      OR      M606
      OUT     M606
7648  LD      M605
      OR      M607
      ANI     M606
      ANI     M126
      ANI     M164
      ANI     M206
      ANI     M1053
      ANI     M804
      OUT     M607
7657  LD      X14  ; Ax#1 Positioning completed
      OR      M609
      AND     M606
      OUT     M609
      LD      B0A2
      OR      M608
      ANB
      OUT     M608
7665  MCR     N0
7666  LDI     M600
      OUT     M610
7668  LD      M600
      ANI     M608
      ANI     M582
      ANI     M584
      LD      M550
      ANI     M558
      ORB
      OR      M410
      OR      M411
      OR      M122
      OUT     M615
7679  LD      M615
      AND     Y67  ; GFC vise/clamp
      OUT     M616
      OUT     T59 K5
7686  LD      M615
      LD      M617
      AND     M92
      ORB
      ANI     Y67  ; GFC vise/clamp
      ANI     M520
      OUT     M617
      OUT     T60 K5
